ABB RobotStudio station: myGofa_20220204-143653.rsstn

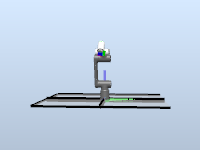
Station myGofa (saved by RobotStudio 21.2.9526.0)
Controller CRB15000_5_95
  mechanical unit ROB_1: CRB15000_5_95__01, 6 joints, base frame (0, 0, 0) mm
Layout (positions relative to the parent item):
  - CRB15000_5_95__01 [mechanism, from Robots\CRB15000_5_95__01.rslib] at (0, 0, 0) mm; joint values [-0.0181, 0.2441, -0.2055, -0.0042, 0.688, -0.2816] (rad or m)
